TYPE stLoadData :
STRUCT
	sLoadID: STRING[30];
	rRig1_LoadDemand:REAL;
	rRig2_LoadDemand:REAL;
	rRig3_LoadDemand:REAL;
	rPitchAngleDemand:REAL;
	bStart:BOOL;
	bConnect:BOOL;
	bHeartbeat:BOOL;
END_STRUCT
END_TYPE

(* stored: Version 1.1.0.1, ProductVersion 3.1.4024.9
   DUT stLoadData: Id {09dff953-6f73-43d0-98d9-ec67810ee5ab} *)
